// TIA Portal V17 export
// export: Created 2023-12-22T15:03:03.4183449Z, ExportSetting WithDefaults, DisplayName Totally Integrated Automation Portal, DisplayVersion V17, DisplayName TIA Portal Openness, DisplayVersion V17, DisplayName TIA Portal Version Control Interface, DisplayVersion V17, DisplayName STEP 7 Professional, DisplayVersion V17, DisplayName STEP 7 Safety, DisplayVersion V17, DisplayName WinCC Advanced, DisplayVersion V17
DATA_BLOCK "DIx_1_DB"   // DB200
VERSION : 0.1
// stored: AutoNumber false, DBAccessibleFromOPCUA true, DBAccessibleFromWebserver true, InstanceOfName DIx_1, InstanceOfType FB
"DIx_1"
   // VAR RETAIN
   //    AllBlock { S7_SetPoint := 'True'} : "DI_ex";
   //    RM_impulse { S7_SetPoint := 'True'} : "DI_ex";
   //    "3Fok" { S7_SetPoint := 'True'} : "DI_ex";
   //    signal_4 { S7_SetPoint := 'True'} : "DI_ex";
   //    signal_5 { S7_SetPoint := 'True'} : "DI_ex";
   //    signal_6 { S7_SetPoint := 'True'} : "DI_ex";
   //    signal_7 { S7_SetPoint := 'True'} : "DI_ex";
   //    signal_8 { S7_SetPoint := 'True'} : "DI_ex";
   //    signal_9 { S7_SetPoint := 'True'} : "DI_ex";
   //    signal_10 { S7_SetPoint := 'True'} : "DI_ex";
   //    signal_11 { S7_SetPoint := 'True'} : "DI_ex";
   //    signal_12 { S7_SetPoint := 'True'} : "DI_ex";
   //    Time_DTL { S7_SetPoint := 'True'} : DTL := DTL#2023-05-02-18:36:48.766257666;
   // END_VAR
BEGIN
   AllBlock.Use.Inverse := FALSE;
   AllBlock.Use.Indirect := TRUE;
   AllBlock.ADDR_Byte := 0;
   AllBlock.ADDR_Bit := 0;
   AllBlock.Filter_On.SP := 16#02;
   AllBlock.Filter_Off.SP := 16#02;
   RM_impulse.Use.Inverse := FALSE;
   RM_impulse.Use.Indirect := TRUE;
   RM_impulse.ADDR_Byte := 0;
   RM_impulse.ADDR_Bit := 1;
   RM_impulse.Filter_On.SP := 16#02;
   RM_impulse.Filter_Off.SP := 16#02;
   "3Fok".Use.Inverse := FALSE;
   "3Fok".Use.Indirect := TRUE;
   "3Fok".ADDR_Byte := 0;
   "3Fok".ADDR_Bit := 2;
   "3Fok".Filter_On.SP := 16#02;
   "3Fok".Filter_Off.SP := 16#02;
   signal_4.Use.Inverse := FALSE;
   signal_4.Use.Indirect := TRUE;
   signal_4.ADDR_Byte := 0;
   signal_4.ADDR_Bit := 9;
   signal_4.Filter_On.SP := 16#02;
   signal_4.Filter_Off.SP := 16#02;
   signal_5.Use.Inverse := FALSE;
   signal_5.Use.Indirect := TRUE;
   signal_5.ADDR_Byte := 0;
   signal_5.ADDR_Bit := 9;
   signal_5.Filter_On.SP := 16#02;
   signal_5.Filter_Off.SP := 16#02;
   signal_6.Use.Inverse := FALSE;
   signal_6.Use.Indirect := TRUE;
   signal_6.ADDR_Byte := 0;
   signal_6.ADDR_Bit := 9;
   signal_6.Filter_On.SP := 16#02;
   signal_6.Filter_Off.SP := 16#02;
   signal_7.Use.Inverse := FALSE;
   signal_7.Use.Indirect := TRUE;
   signal_7.ADDR_Byte := 0;
   signal_7.ADDR_Bit := 9;
   signal_7.Filter_On.SP := 16#02;
   signal_7.Filter_Off.SP := 16#02;
   signal_8.Use.Inverse := FALSE;
   signal_8.Use.Indirect := TRUE;
   signal_8.ADDR_Byte := 0;
   signal_8.ADDR_Bit := 9;
   signal_8.Filter_On.SP := 16#02;
   signal_8.Filter_Off.SP := 16#02;
   signal_9.Use.Inverse := FALSE;
   signal_9.Use.Indirect := TRUE;
   signal_9.ADDR_Byte := 0;
   signal_9.ADDR_Bit := 9;
   signal_9.Filter_On.SP := 16#02;
   signal_9.Filter_Off.SP := 16#02;
   signal_10.Use.Inverse := FALSE;
   signal_10.Use.Indirect := TRUE;
   signal_10.ADDR_Byte := 0;
   signal_10.ADDR_Bit := 9;
   signal_10.Filter_On.SP := 16#02;
   signal_10.Filter_Off.SP := 16#02;
   signal_11.Use.Inverse := FALSE;
   signal_11.Use.Indirect := TRUE;
   signal_11.ADDR_Byte := 0;
   signal_11.ADDR_Bit := 9;
   signal_11.Filter_On.SP := 16#02;
   signal_11.Filter_Off.SP := 16#02;
   signal_12.Use.Inverse := FALSE;
   signal_12.Use.Indirect := TRUE;
   signal_12.ADDR_Byte := 0;
   signal_12.ADDR_Bit := 9;
   signal_12.Filter_On.SP := 16#02;
   signal_12.Filter_Off.SP := 16#02;
END_DATA_BLOCK
